TYPE "LogInOut_ShW"
VERSION : 0.1
   STRUCT
      Trigger : Bool;
      OperatorNo : String[48];
      Result : Int;
      Completed : Bool;
   END_STRUCT;

END_TYPE

